Universal Robots URScript: Program_Control_Move_Predetermined.script

def Program_Template():
   set_standard_analog_input_domain(0, 1)
   set_standard_analog_input_domain(1, 1)
   set_tool_analog_input_domain(0, 1)
   set_tool_analog_input_domain(1, 1)
   set_analog_outputdomain(0, 0)
   set_analog_outputdomain(1, 0)
   set_tool_voltage(0)
   set_input_actions_to_default()
   set_tcp(p[0.0,0.0,0.0,0.0,0.0,0.0])
   set_payload(0.0)
   set_gravity([0.0, 0.0, 9.82])
   global Base=p[0.0,0.0,0.0,0.0,0.0,0.0]
   rtde_set_watchdog("speed_slider_mask", 10.0, "ignore")
   global setp = [0,0,0,0,0,0]
   global move = [0,0,0,0]




	movej([-1.378465,-0.727069,0.285923,-0.152539,1.570796,-1.477043],0.200000,0.200000,0.000000,0.000000)
	movej([-1.570697,-1.054600,0.571733,-0.109435,1.315900,-1.402730],0.200000,0.200000,0.000000,0.029461)
	movej([-1.749022,-1.355698,0.865940,-0.256523,1.301870,-1.329885],0.200000,0.200000,0.000000,0.027657)
	movej([-1.969825,-1.621292,1.080726,-0.360678,1.287112,-1.230906],0.200000,0.200000,0.000000,0.026038)
	movej([-2.273219,-1.884406,1.272629,-0.451082,1.267885,-1.078859],0.200000,0.200000,0.000000,0.024819)
	movej([-2.565963,-2.101823,1.643192,-1.112165,1.570796,-0.938121],0.200000,0.200000,0.000000,0.024195)
	movej([-3.280186,-2.395905,1.736986,-0.911877,1.570796,-0.062791],0.200000,0.200000,0.000000,0.024275)
	movej([-4.216986,-2.545082,1.936708,-1.064801,1.570796,1.032809],0.200000,0.200000,0.000000,0.025046)
	movej([-4.822558,-2.573293,2.107753,-1.170387,1.570796,1.802269],0.200000,0.200000,0.000000,0.026373)
	movej([-4.968647,-2.416467,2.277822,-1.432151,1.570796,2.108992],0.200000,0.200000,0.000000,0.028052)
	movej([-5.012341,-1.935852,2.397614,-2.032558,1.570796,2.313794],0.200000,0.200000,0.000000,0.029868)
	movej([-5.079407,-1.358079,2.308383,-2.521101,1.570796,2.541967],0.200000,0.200000,0.000000,0.031626)
	movej([-5.154469,-0.858545,2.018272,-2.730523,1.570796,2.778136],0.200000,0.200000,0.000000,0.033169)
	movej([-5.233275,-0.424447,1.565183,-2.711532,1.570796,3.018049],0.200000,0.200000,0.000000,0.034375)

  textmsg("Ending MoveJ")



end
